PROGRAM SAFETY


//IF GVL_Safety.RUN_STOP = TRUE THEN

//	IF GVL_Safety.SAFETY_Permission = FALSE THEN
	
//		CASE GVL_Safety.SafetySate OF
		
//			0:
//				GVL_Safety.ErrorAck := FALSE;
//				GVL_Safety.SafetySate := GVL_Safety.SafetySate + 10;
//			10:
//				GVL_Safety.ErrorAck := TRUE;
//				GVL_Safety.SafetySate := GVL_Safety.SafetySate + 10;
//			20:
//				GVL_Safety.ErrorAck := FALSE;
//				GVL_Safety.SafetySate := GVL_Safety.SafetySate + 10;
//			30:		
//				GVL_Safety.AX5805_ErrACK := FALSE;
//				GVL_Safety.SafetySate := GVL_Safety.SafetySate + 10;
//			40:	
//				GVL_Safety.AX5805_ErrACK := TRUE;
//				GVL_Safety.SafetySate := GVL_Safety.SafetySate + 10;
//			50:
//				GVL_Safety.AX5805_ErrACK := FALSE;
//				GVL_Safety.SafetySate := GVL_Safety.SafetySate + 10;	
//			60:
//				GVL_Safety.RestartFBs_TSG := FALSE;
//				GVL_Safety.SafetySate := GVL_Safety.SafetySate + 10;
//			70:
//				GVL_Safety.RestartFBs_TSG := TRUE;
//				GVL_Safety.SafetySate := GVL_Safety.SafetySate + 10;	
//			80:
//				GVL_Safety.RestartFBs_TSG := FALSE;
//				GVL_Safety.SafetySate := GVL_Safety.SafetySate + 10;	
//			90:		
//				GVL_Safety.SafetySate := 0;

//		END_CASE
//	END_IF	

//END_IF

END_PROGRAM

(* stored: Version 1.1.0.1, ProductVersion 3.1.4024.15
   POU SAFETY: Id {fe3eb017-1e4d-407b-90fe-7196ffdfbcaf}, SpecialFunc None *)
